// TIA Portal V17 export
// export: Created 2026-04-12T10:31:03.2037994Z, ExportSetting WithDefaults, DisplayName Totally Integrated Automation Portal, DisplayVersion V17 Update 4, DisplayName TIA Portal Openness, DisplayVersion V17 Update 4, DisplayName TIA Portal Version Control Interface, DisplayVersion V17, DisplayName SINAMICS Startdrive Advanced, DisplayVersion V17, DisplayName SINAMICS Startdrive G130, G150, S120, S150, SINAMICS MV, S210, DisplayVersion V17, DisplayName SINAMICS Startdrive G110M, G120, G120C, G120D, G120P, G115D, DisplayVersion V17, DisplayName STEP 7 Professional, DisplayVersion V17 Update 4, DisplayName STEP 7 Safety, DisplayVersion V17, DisplayName WinCC Advanced, DisplayVersion V17 Update 4
ORGANIZATION_BLOCK "Main"   // OB1, LAD, ProgramCycle
TITLE = "Main Program Sweep (Cycle)"
{ S7_Optimized_Access := 'TRUE' }
VERSION : 0.1
// stored: AutoNumber true, IsIECCheckEnabled false, SetENOAutomatically false
   VAR_INPUT
      Initial_Call : Bool;   // Initial call of this OB
      Remanence : Bool;   // =True, if remanent data are available
   END_VAR
BEGIN

REGION Network 1
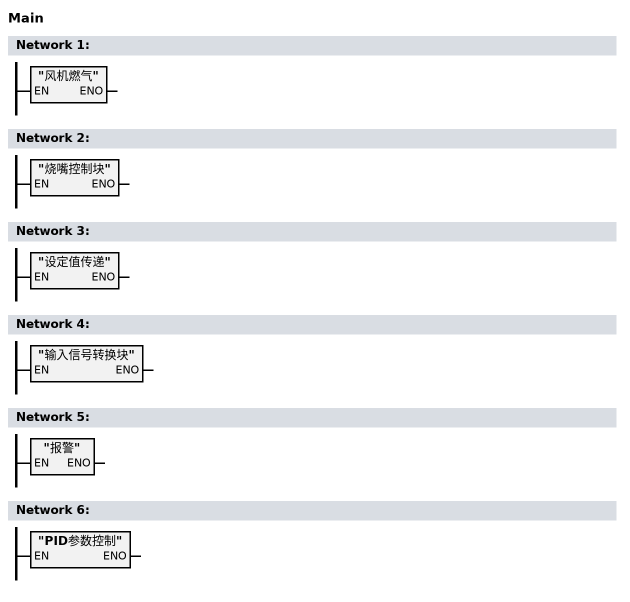
   RUNG wire#powerrail
      "风机燃气"()
   END_RUNG
   // the same network as SCL:
   "风机燃气"();
END_REGION

REGION Network 2
   RUNG wire#powerrail
      "烧嘴控制块"()
   END_RUNG
   // the same network as SCL:
   "烧嘴控制块"();
END_REGION

REGION Network 3
   RUNG wire#powerrail
      "设定值传递"()
   END_RUNG
   // the same network as SCL:
   "设定值传递"();
END_REGION

REGION Network 4
   RUNG wire#powerrail
      "输入信号转换块"()
   END_RUNG
   // the same network as SCL:
   "输入信号转换块"();
END_REGION

REGION Network 5
   RUNG wire#powerrail
      "报警"()
   END_RUNG
   // the same network as SCL:
   "报警"();
END_REGION

REGION Network 6
   RUNG wire#powerrail
      "PID参数控制"()
   END_RUNG
   // the same network as SCL:
   "PID参数控制"();
END_REGION
END_ORGANIZATION_BLOCK
